(* Logix 5000 project; controller Reto2 Emulate 5570 rev 30.12; software revision 30.00 *)

TASK MainTask (continuous, watchdog 500 ms) : MainProgram

MODULES
   Local : Emulate 5570 (ICP 2, rev 30.12)
END_MODULES

VAR_GLOBAL   (* controller tags *)
   ActLX : INT;
   ActLY : INT;
   B1 : BOOL;
   B2A : BOOL;
   B2B : BOOL;
   CilinderMax : BOOL;
   CilinderMin : BOOL;
   CilinderPos : INT;
   FillerMax : BOOL;
   FillerMin : BOOL;
   FillerPos : INT;
   Manguera : BOOL;
   P : BOOL;   // Selector de baldosas
   S1 : BOOL;
   S2 : BOOL;
   SourceTiles : BOOL;
   Start : BOOL;
   SXmax : BOOL;
   SXmin : BOOL;
   TileMax : BOOL;
   TileMin : BOOL;
   TilePos : INT;
   VelX : INT;
   VelY : INT;
   Ymax : BOOL;
   Ymin : BOOL;
END_VAR

PROGRAM MainProgram   (* main routine MainRoutine *)
VAR
   Action_000 : SFC_ACTION := (Status := 16#0020_0000, PauseTimer := 1);
   Action_001 : SFC_ACTION := (Status := 16#0020_0000, PauseTimer := 1);
   Action_002 : SFC_ACTION := (Status := 16#0020_0000, PauseTimer := 1);
   Action_003 : SFC_ACTION := (Status := 16#0020_0000, PauseTimer := 1);
   Action_004 : SFC_ACTION := (Status := 16#0020_0000, PauseTimer := 1);
   Action_005 : SFC_ACTION := (Status := 16#0020_0000, PauseTimer := 1);
   Action_006 : SFC_ACTION := (Status := 16#0020_0000, PauseTimer := 1);
   Action_007 : SFC_ACTION := (Status := 16#0020_0000, PauseTimer := 1);
   Action_008 : SFC_ACTION := (Status := 16#0020_0000, PauseTimer := 1);
   Action_009 : SFC_ACTION := (Status := 16#0020_0000, PauseTimer := 1);
   Action_010 : SFC_ACTION := (Status := 16#0020_0000, PauseTimer := 1);
   Action_011 : SFC_ACTION := (Status := 16#0020_0000, PauseTimer := 1);
   Action_012 : SFC_ACTION := (Status := 16#0020_0000, PauseTimer := 1);
   Action_013 : SFC_ACTION := (Status := 16#0020_0000, PauseTimer := 1);
   Action_014 : SFC_ACTION := (Status := 16#0020_0000, PauseTimer := 1);
   Action_015 : SFC_ACTION := (Status := 16#0020_0000, PauseTimer := 1);
   Action_016 : SFC_ACTION := (Status := 16#0020_0000, PauseTimer := 1);
   Action_017 : SFC_ACTION := (Status := 16#0020_0000, PauseTimer := 1);
   Action_018 : SFC_ACTION := (Status := 16#0020_0000, PauseTimer := 1);
   Action_019 : SFC_ACTION := (Status := 16#0020_0000, PauseTimer := 1);
   Action_020 : SFC_ACTION := (Status := 16#0020_0000, PauseTimer := 1);
   Action_021 : SFC_ACTION := (Status := 16#0020_0000, PauseTimer := 1);
   C1 : COUNTER := (PRE := 4);
   C2 : COUNTER := (PRE := 4);
   ResetC1 : BOOL;
   ResetC2 : BOOL;
   StartPress : BOOL;
   Step_000 : SFC_STEP := (Status := 16#0020_0000, PauseTimer := 1);
   Step_001 : SFC_STEP := (Status := 16#0020_0000, PauseTimer := 1);
   Step_002 : SFC_STEP := (Status := 16#0020_0000, PauseTimer := 1);
   Step_003 : SFC_STEP := (Status := 16#0020_0000, PauseTimer := 1);
   Step_004 : SFC_STEP := (Status := 16#0020_0000, PauseTimer := 1);
   Step_005 : SFC_STEP := (Status := 16#0020_0000, PauseTimer := 1);
   Step_006 : SFC_STEP := (Status := 16#0020_0000, PauseTimer := 1);
   Step_007 : SFC_STEP := (Status := 16#0020_0000, PauseTimer := 1);
   Step_008 : SFC_STEP := (Status := 16#0020_0000, PauseTimer := 1, T := 100);
   Step_009 : SFC_STEP := (Status := 16#0020_0000, PauseTimer := 1);
   Step_010 : SFC_STEP := (Status := 16#0020_0000, PauseTimer := 1);
   Step_011 : SFC_STEP := (Status := 16#0020_0000, PauseTimer := 1);
   Step_012 : SFC_STEP := (Status := 16#0020_0000, PauseTimer := 1);
   Step_013 : SFC_STEP := (Status := 16#0020_0000, PauseTimer := 1);
   Step_014 : SFC_STEP := (Status := 16#0020_0000, PauseTimer := 1);
   Step_015 : SFC_STEP := (Status := 16#0020_0000, PauseTimer := 1);
   Step_016 : SFC_STEP := (Status := 16#0020_0000, PauseTimer := 1);
   Step_017 : SFC_STEP := (Status := 16#0020_0000, PauseTimer := 1);
   Step_018 : SFC_STEP := (Status := 16#0020_0000, PauseTimer := 1);
   Step_019 : SFC_STEP := (Status := 16#0020_0000, PauseTimer := 1);
   Step_020 : SFC_STEP := (Status := 16#0020_0000, PauseTimer := 1);
   Step_021 : SFC_STEP := (Status := 16#0020_0000, PauseTimer := 1);
   Step_022 : SFC_STEP := (Status := 16#0020_0000, PauseTimer := 1);
   Step_023 : SFC_STEP := (Status := 16#0020_0000, PauseTimer := 1);
   Step_024 : SFC_STEP := (Status := 16#0020_0000, PauseTimer := 1);
   Step_025 : SFC_STEP := (Status := 16#0020_0000, PauseTimer := 1);
   Step_026 : SFC_STEP := (Status := 16#0020_0000, PauseTimer := 1);
   Step_027 : SFC_STEP := (Status := 16#0020_0000, PauseTimer := 1);
   Step_028 : SFC_STEP := (Status := 16#0020_0000, PauseTimer := 1);
   Step_029 : SFC_STEP := (Status := 16#0020_0000, PauseTimer := 1);
   Step_030 : SFC_STEP := (Status := 16#0020_0000, PauseTimer := 1);
   Step_031 : SFC_STEP := (Status := 16#0020_0000, PauseTimer := 1);
   Step_032 : SFC_STEP := (Status := 16#0020_0000, PauseTimer := 1);
   Step_033 : SFC_STEP := (Status := 16#0020_0000, PauseTimer := 1);
   Step_034 : SFC_STEP := (Status := 16#0020_0000, PauseTimer := 1);
   Step_035 : SFC_STEP := (Status := 16#0020_0000, PauseTimer := 1);
   Step_036 : SFC_STEP := (Status := 16#0020_0000, PauseTimer := 1);
   Step_037 : SFC_STEP := (Status := 16#0020_0000, PauseTimer := 1);
   Step_038 : SFC_STEP := (Status := 16#0020_0000, PauseTimer := 1);
   Step_040 : SFC_STEP := (Status := 16#0020_0000, PauseTimer := 1);
   Step_041 : SFC_STEP := (Status := 16#0020_0000, PauseTimer := 1);
   Step_042 : SFC_STEP := (Status := 16#0020_0000, PauseTimer := 1);
   Step_050 : SFC_STEP := (Status := 16#0020_0000, PauseTimer := 1, PRE := 200);
   Stop_000 : SFC_STOP;
   Test : BOOL;
   Tran_000 : BOOL;
   Tran_001 : BOOL;
   Tran_002 : BOOL;
   Tran_003 : BOOL;
   Tran_004 : BOOL;
   Tran_005 : BOOL;
   Tran_006 : BOOL;
   Tran_007 : BOOL;
   Tran_008 : BOOL;
   Tran_009 : BOOL;
   Tran_010 : BOOL;
   Tran_011 : BOOL;
   Tran_012 : BOOL;
   Tran_013 : BOOL;
   Tran_014 : BOOL;
   Tran_015 : BOOL;
   Tran_016 : BOOL;
   Tran_017 : BOOL;
   Tran_018 : BOOL;
   Tran_019 : BOOL;
   Tran_020 : BOOL;
   Tran_021 : BOOL;
   Tran_022 : BOOL;
   Tran_023 : BOOL;
   Tran_024 : BOOL;
   Tran_025 : BOOL;
   Tran_026 : BOOL;
   Tran_027 : BOOL;
   Tran_028 : BOOL;
   Tran_029 : BOOL;
   Xmin_T : BOOL;
END_VAR

ROUTINE BetterPress   (* sequential function chart *)
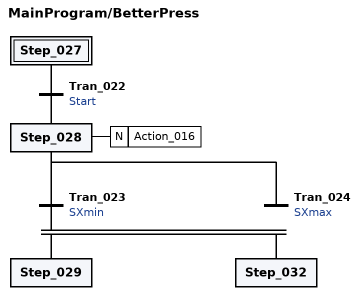
   INITIAL_STEP Step_027:
   END_STEP
   TRANSITION Tran_022 FROM Step_027 TO Step_028
      := Start
         
   END_TRANSITION
   STEP Step_028:
      ACTION Action_016 (N):
         Manguera :=1;
         
      END_ACTION
   END_STEP
   TRANSITION Tran_023 FROM Step_028 TO (Step_032, Step_029)
      := SXmin
         
   END_TRANSITION
   TRANSITION Tran_024 FROM Step_028 TO ()
      := SXmax
         
   END_TRANSITION
   STEP Step_029:
   END_STEP
   STEP Step_032:
   END_STEP
END_ROUTINE

ROUTINE LD_Bandas   (* ladder *)
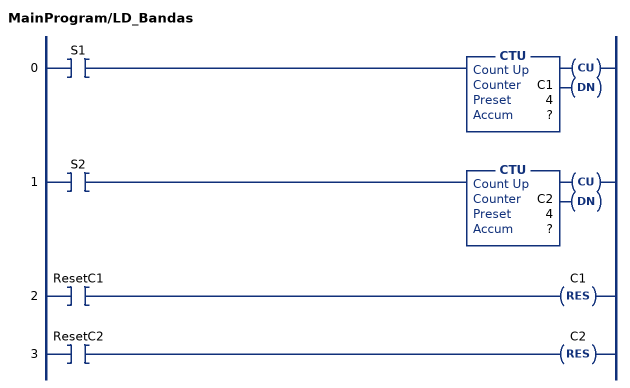
   0: XIC(S1)CTU(C1,?,?);
   1: XIC(S2)CTU(C2,?,?);
   2: XIC(ResetC1)RES(C1);
   3: XIC(ResetC2)RES(C2);
END_ROUTINE

ROUTINE MainRoutine   (* ladder *)
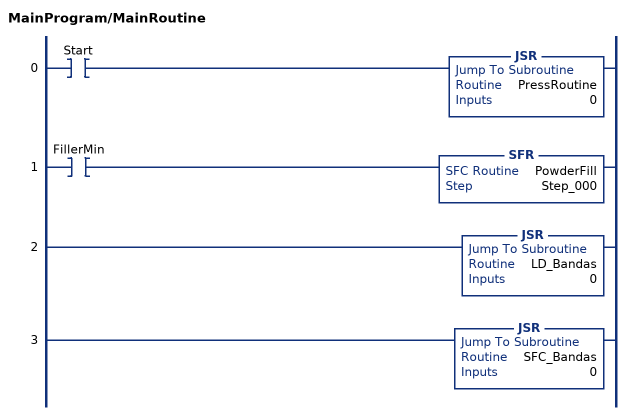
   0: XIC(Start)JSR(PressRoutine,0);
   1: XIC(FillerMin)SFR(PowderFill,Step_000);
   2: JSR(LD_Bandas,0);
   3: JSR(SFC_Bandas,0);
END_ROUTINE

ROUTINE PowderFill   (* sequential function chart *)
// Ceramic Press Logic
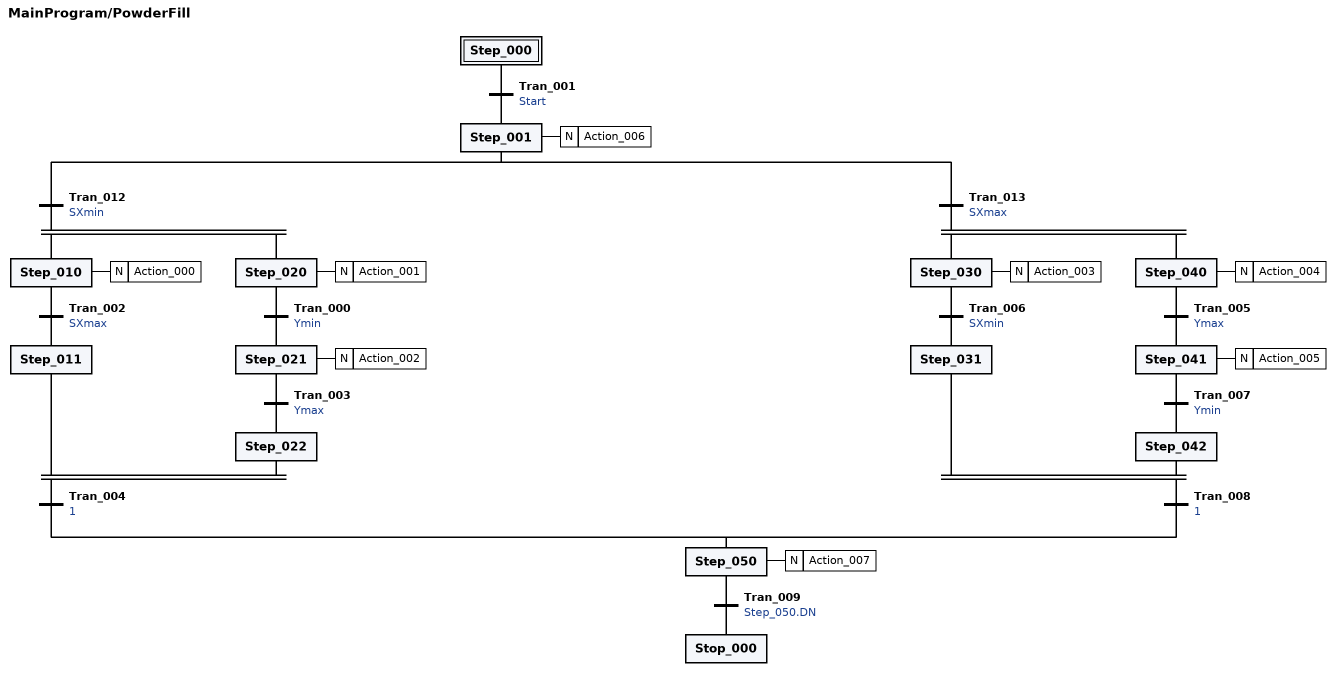
   INITIAL_STEP Step_000:
   END_STEP
   TRANSITION Tran_001 FROM Step_000 TO Step_001
      := Start
   END_TRANSITION
   STEP Step_001:
      ACTION Action_006 (N):
         Manguera :=1;
      END_ACTION
   END_STEP
   TRANSITION Tran_012 FROM Step_001 TO (Step_020, Step_010)
      := SXmin
   END_TRANSITION
   TRANSITION Tran_013 FROM Step_001 TO (Step_040, Step_030)
      := SXmax
   END_TRANSITION
   STEP Step_010:
      ACTION Action_000 (N):
         ActLX := 1220;
      END_ACTION
   END_STEP
   STEP Step_020:
      ACTION Action_001 (N):
         ActLY := 0;
      END_ACTION
   END_STEP
   STEP Step_030:
      ACTION Action_003 (N):
         ActLX := 0;
      END_ACTION
   END_STEP
   STEP Step_040:
      ACTION Action_004 (N):
         ActLY := 710;
      END_ACTION
   END_STEP
   TRANSITION Tran_002 FROM Step_010 TO Step_011
      := SXmax
   END_TRANSITION
   TRANSITION Tran_000 FROM Step_020 TO Step_021
      := Ymin
   END_TRANSITION
   TRANSITION Tran_006 FROM Step_030 TO Step_031
      := SXmin
   END_TRANSITION
   TRANSITION Tran_005 FROM Step_040 TO Step_041
      := Ymax
   END_TRANSITION
   STEP Step_021:
      ACTION Action_002 (N):
         ActLY := 710;
         
      END_ACTION
   END_STEP
   STEP Step_041:
      ACTION Action_005 (N):
         ActLY := 0;
      END_ACTION
   END_STEP
   TRANSITION Tran_003 FROM Step_021 TO Step_022
      := Ymax
   END_TRANSITION
   TRANSITION Tran_007 FROM Step_041 TO Step_042
      := Ymin
   END_TRANSITION
   STEP Step_011:
   END_STEP
   STEP Step_022:
   END_STEP
   STEP Step_031:
   END_STEP
   STEP Step_042:
   END_STEP
   TRANSITION Tran_004 FROM (Step_011, Step_022) TO Step_050
      := 1
   END_TRANSITION
   TRANSITION Tran_008 FROM (Step_031, Step_042) TO Step_050
      := 1
   END_TRANSITION
   STEP Step_050:
      ACTION Action_007 (N):
         Manguera :=0;
      END_ACTION
   END_STEP
   TRANSITION Tran_009 FROM Step_050 TO Stop_000
      := Step_050.DN
   END_TRANSITION
   STOP Stop_000;
END_ROUTINE

ROUTINE PressRoutine   (* sequential function chart *)
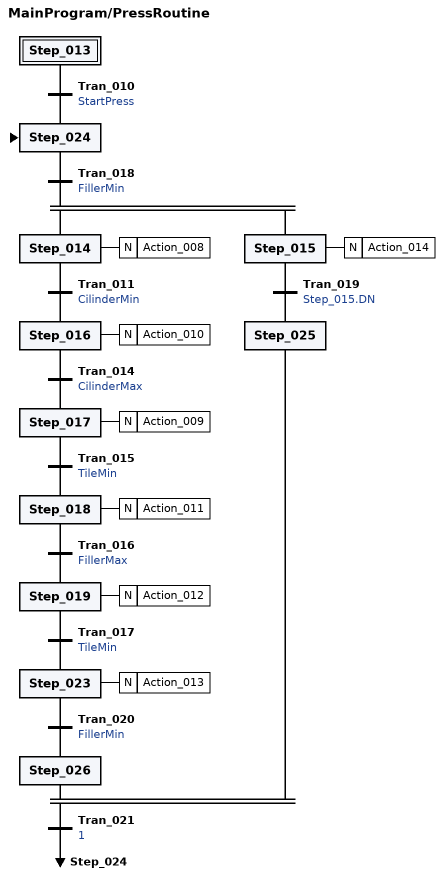
   INITIAL_STEP Step_013:
   END_STEP
   TRANSITION Tran_010 FROM Step_013 TO Step_024
      := StartPress
   END_TRANSITION
   STEP Step_024:
   END_STEP
   TRANSITION Tran_018 FROM Step_024 TO (Step_015, Step_014)
      := FillerMin
   END_TRANSITION
   STEP Step_014:
      ACTION Action_008 (N):
         CilinderPos :=0;
         SourceTiles :=1;
      END_ACTION
   END_STEP
   STEP Step_015:
      ACTION Action_014 (N):
         JSR(PowderFill,1,Start,Step_050.DN);
      END_ACTION
   END_STEP
   TRANSITION Tran_011 FROM Step_014 TO Step_016
      := CilinderMin
         
   END_TRANSITION
   TRANSITION Tran_019 FROM Step_015 TO Step_025
      := Step_015.DN
         
   END_TRANSITION
   STEP Step_016:
      ACTION Action_010 (N):
         SourceTiles :=0;
         CilinderPos := 140;
      END_ACTION
   END_STEP
   TRANSITION Tran_014 FROM Step_016 TO Step_017
      := CilinderMax
   END_TRANSITION
   STEP Step_017:
      ACTION Action_009 (N):
         TilePos := 9.5;
      END_ACTION
   END_STEP
   TRANSITION Tran_015 FROM Step_017 TO Step_018
      := TileMin
         
   END_TRANSITION
   STEP Step_018:
      ACTION Action_011 (N):
         FillerPos := 800;
      END_ACTION
   END_STEP
   TRANSITION Tran_016 FROM Step_018 TO Step_019
      := FillerMax
   END_TRANSITION
   STEP Step_019:
      ACTION Action_012 (N):
         TilePos := 0;
      END_ACTION
   END_STEP
   TRANSITION Tran_017 FROM Step_019 TO Step_023
      := TileMin
         
   END_TRANSITION
   STEP Step_023:
      ACTION Action_013 (N):
         FillerPos := 0;
      END_ACTION
   END_STEP
   TRANSITION Tran_020 FROM Step_023 TO Step_026
      := FillerMin
         
   END_TRANSITION
   STEP Step_026:
   END_STEP
   STEP Step_025:
   END_STEP
   TRANSITION Tran_021 FROM (Step_026, Step_025) TO Step_024
      := 1
         
   END_TRANSITION
END_ROUTINE

ROUTINE SFC_Bandas   (* sequential function chart *)
// Logica para mover las bandas entre maquinas
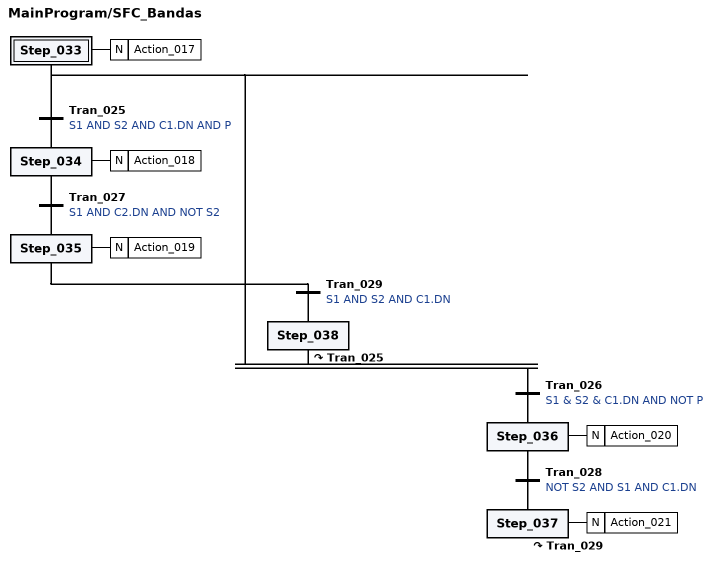
   INITIAL_STEP Step_033:
      ACTION Action_017 (N):
         B1 := 1;
         B2A := 1;
         B2B := 0;
      END_ACTION
   END_STEP
   TRANSITION Tran_025 FROM (Step_033, Step_038) TO Step_034
      := S1 AND S2 AND C1.DN AND P
   END_TRANSITION
   TRANSITION Tran_026 FROM (Step_033, Step_038) TO Step_036
      := S1 & S2 & C1.DN AND NOT P
   END_TRANSITION
   STEP Step_034:
      ACTION Action_018 (N):
         B1 :=0;
         B2A :=1;
         B2B :=0;
      END_ACTION
   END_STEP
   STEP Step_036:
      ACTION Action_020 (N):
         B1 :=0;
         B2A :=0;
         B2B :=1;
      END_ACTION
   END_STEP
   TRANSITION Tran_027 FROM Step_034 TO Step_035
      := S1 AND C2.DN AND NOT S2
   END_TRANSITION
   TRANSITION Tran_028 FROM Step_036 TO Step_037
      := NOT S2 AND S1 AND C1.DN
   END_TRANSITION
   STEP Step_035:
      ACTION Action_019 (N):
         ResetC1 := 1;
         B1 := 1;
         B2A := 1;
         ResetC1 := 0;
      END_ACTION
   END_STEP
   STEP Step_037:
      ACTION Action_021 (N):
         ResetC1 := 1;
         B1 := 1;
         B2A := 1;
         ResetC1 := 0;
      END_ACTION
   END_STEP
   TRANSITION Tran_029 FROM (Step_037, Step_035) TO Step_038
      := S1 AND S2 AND C1.DN
   END_TRANSITION
   STEP Step_038:
   END_STEP
END_ROUTINE
END_PROGRAM
